FUNCTION_BLOCK FB_Coche EXTENDS FB_Vehiculo
VAR_INPUT
	velocidadMaxima : REAL;
END_VAR
VAR_OUTPUT
END_VAR
VAR
END_VAR

METHOD getVelocidadMaxima : REAL
VAR_INPUT
END_VAR
getVelocidadMaxima := velocidadMaxima;
END_METHOD

END_FUNCTION_BLOCK

(* stored: Version 1.1.0.1, ProductVersion 3.1.4024.12
   POU FB_Coche: Id {e23fc4b7-6214-4b36-a282-d7ecb2ef8288}, SpecialFunc None
   Method getVelocidadMaxima: Id {4aeecc75-7896-4a31-a0db-277b1fbade77} *)
